FUNCTION_BLOCK FB_Ergonomics EXTENDS FB_StateMachine IMPLEMENTS I_StateMachine
VAR_INPUT
	bStart : BOOL;
	fbStepper : REFERENCE TO FB_Stepper;
	fbLinearActuator : REFERENCE TO FB_LinearActuator;
	
END_VAR
VAR
	eInnerState : E_ErgonomicStates;
//	bCompleted : BOOL;
//	dtTimeCompleted: DATE_AND_TIME;
	stErgoCommands :  ST_ErgoCommands;
END_VAR

OuterLopSM();

METHOD Disable : BOOL
fbStepper.Active:=FALSE;
fbLinearActuator.Active:=FALSE;

Disable := TRUE;
END_METHOD

PROPERTY ErgoCommands : ST_ErgoCommands
GET
ErgoCommands := stErgoCommands;
END_GET
SET
THIS^.stErgoCommands := ErgoCommands;
END_SET
END_PROPERTY

METHOD InnerLoopSM : BOOL
// update all children FBs

CASE CyclicInnerCase(TO_STRING(eInnerState)) OF
	E_ErgonomicStates.Idle:
		IF bStart THEN
			bStart := FALSE;
			ChangeInnerState(E_ErgonomicStates.WaitForCommand);
		END_IF
	
	E_ErgonomicStates.WaitForCommand:
		IF stErgoCommands.Done THEN
			ChangeInnerState(E_ErgonomicStates.Idle);
		END_IF
		
	E_ErgonomicStates.JogLeftStepperOut:
		ChangeInnerState(E_ErgonomicStates.WaitForCommand);
		
	E_ErgonomicStates.JogLeftStepperIn:
		ChangeInnerState(E_ErgonomicStates.WaitForCommand);		
		
	E_ErgonomicStates.JogRightStepperOut:
		ChangeInnerState(E_ErgonomicStates.WaitForCommand);
		
	E_ErgonomicStates.JogRightStepperIn:
		ChangeInnerState(E_ErgonomicStates.WaitForCommand);	
		
	E_ErgonomicStates.JogLeftLinActuatorUp:
		ChangeInnerState(E_ErgonomicStates.WaitForCommand);
		
	E_ErgonomicStates.JogLeftLinActuatorDown:
		ChangeInnerState(E_ErgonomicStates.WaitForCommand);
		
	E_ErgonomicStates.JogRightLinActuatorUp:
		ChangeInnerState(E_ErgonomicStates.WaitForCommand);
		
	E_ErgonomicStates.JogRightLinActuatorDown:
		ChangeInnerState(E_ErgonomicStates.WaitForCommand);
		
END_CASE
END_METHOD

METHOD Reset : BOOL
//bCompleted := FALSE;
//dtTimeCompleted := DATE_AND_TIME#1970-1-1-0:0:0;
END_METHOD

METHOD Setup : BOOL
eStateMachineSourceID := eStateSourceID;
SetInnerEnumeration(nStateEnum:=THIS^.eInnerState);
END_METHOD

PROPERTY Waiting : BOOL
GET
Waiting := (eInnerState = E_ErgonomicStates.WaitForCommand);
END_GET
END_PROPERTY

END_FUNCTION_BLOCK

(* stored: Version 1.1.0.1, ProductVersion 3.1.4024.12
   POU FB_Ergonomics: Id {6993645b-63dd-4730-9789-181f704dc6ec}, SpecialFunc None
   Folder Properties: Id {58194c6f-b433-4e17-a779-fcd066af53f1}
   Method Disable: Id {190982a1-4db5-42cc-8726-74036ccb0b0d}
   Property ErgoCommands: Id {3ae45f7d-be97-44eb-9415-91282f532b17}
   Get Get: Id {0ecbe159-97ac-4acf-8c5b-8dda58ce1507}
   Set Set: Id {42834955-cbee-4e6d-b64e-6d9e46ac952f}
   Method InnerLoopSM: Id {891b181b-eec5-45e2-b5a3-cd46ced640e2}
   Method Reset: Id {47bca2af-0103-430b-b509-73ae259725be}
   Method Setup: Id {6487ff34-4ccc-4503-95ba-c93d6ec95a42}
   Property Waiting: Id {c721428f-162e-475e-9d9a-a4ee1f9a78ba}
   Get Get: Id {0b92389d-69c5-419c-8725-60d05ee6f105} *)
